FUNCTION_BLOCK Handbetrieb
VAR_INPUT
END_VAR
VAR_OUTPUT
END_VAR
VAR
END_VAR

// NETWORK 1

END_FUNCTION_BLOCK

(* stored: Version 1.1.0.1, ProductVersion 3.1.4024.4
   POU Handbetrieb: Id {20dece89-6b02-438e-9264-5381e2502ba6}, SpecialFunc None *)
